INTERFACE I_LightTowerComponent

// Sets the component state to TRUE.
METHOD Activate
VAR_INPUT
END_VAR
END_METHOD

// Sets the component state to FALSE.
METHOD Deactivate
VAR_INPUT
END_VAR
END_METHOD

// Gets state of the component. TRUE if active, else FALSE.
PROPERTY State : BOOL
GET
END_GET
END_PROPERTY

END_INTERFACE

(* stored: Version 1.1.0.1, ProductVersion 3.1.4024.13
   Itf I_LightTowerComponent: Id {565a0719-8fd5-0e5c-38ed-27694fe06560}
   Method Activate: Id {cc40e103-f929-0ec3-22f2-2ec071d80a27}
   Method Deactivate: Id {6d59e4ed-68f8-0d8c-3c59-3ae523d53295}
   Property State: Id {aadc2ef6-2d88-0fa8-39fc-e5110e96b1b5}
   Get Get: Id {5b9d3ee7-29b9-06e9-2145-2fbc8558ba2b} *)
